Universal Robots PolyScope program: circle_run.urp

Program circle_run (installation=default directory=/programs/usbdisk createdIn=5.12.4.1101661 lastSavedIn=5.12.4.1101661)
Robot Program (runOnlyOnce=true)
  Script file /programs/usbdisk/circle.script
    | def draw_svg():
    |   draw_z = 0.074940
    |   # home
    |   movel(p[0.598550, -0.129200, 0.105150, 2.249000, -2.194000, 0.000000], a=0.8, v=0.25, r=0.0)
    |   # stroke 0 (form id 0): circle
    |   movel(p[0.452368, -0.119322, 0.118080, 2.230000, -2.212000, 0.000000], a=0.8, v=0.25, r=0.0)
    |   movep(p[0.452368, -0.119322, draw_z, 2.230000, -2.212000, 0.000000], a=0.5, v=0.02, r=0.001426)
    |   movep(p[0.452414, -0.116470, draw_z, 2.230000, -2.212000, 0.000000], a=0.5, v=0.02, r=0.002853)
    |   movep(p[0.452720, -0.110772, draw_z, 2.230000, -2.212000, 0.000000], a=0.5, v=0.02, r=0.002855)
    |   movep(p[0.453238, -0.105086, draw_z, 2.230000, -2.212000, 0.000000], a=0.5, v=0.02, r=0.002856)
    |   movep(p[0.453967, -0.099420, draw_z, 2.230000, -2.212000, 0.000000], a=0.5, v=0.02, r=0.002857)
    |   movep(p[0.454907, -0.093783, draw_z, 2.230000, -2.212000, 0.000000], a=0.5, v=0.02, r=0.002859)
    |   movep(p[0.456055, -0.088182, draw_z, 2.230000, -2.212000, 0.000000], a=0.5, v=0.02, r=0.002860)
    |   movep(p[0.457411, -0.082625, draw_z, 2.230000, -2.212000, 0.000000], a=0.5, v=0.02, r=0.002861)
    |   movep(p[0.458973, -0.077120, draw_z, 2.230000, -2.212000, 0.000000], a=0.5, v=0.02, r=0.002862)
    |   movep(p[0.460738, -0.071675, draw_z, 2.230000, -2.212000, 0.000000], a=0.5, v=0.02, r=0.002863)
    |   movep(p[0.462703, -0.066296, draw_z, 2.230000, -2.212000, 0.000000], a=0.5, v=0.02, r=0.002864)
    |   movep(p[0.464867, -0.060993, draw_z, 2.230000, -2.212000, 0.000000], a=0.5, v=0.02, r=0.002865)
    |   movep(p[0.467226, -0.055771, draw_z, 2.230000, -2.212000, 0.000000], a=0.5, v=0.02, r=0.002866)
    |   movep(p[0.469777, -0.050639, draw_z, 2.230000, -2.212000, 0.000000], a=0.5, v=0.02, r=0.002866)
    |   movep(p[0.472516, -0.045604, draw_z, 2.230000, -2.212000, 0.000000], a=0.5, v=0.02, r=0.002867)
    |   movep(p[0.475439, -0.040672, draw_z, 2.230000, -2.212000, 0.000000], a=0.5, v=0.02, r=0.002867)
    |   movep(p[0.478543, -0.035850, draw_z, 2.230000, -2.212000, 0.000000], a=0.5, v=0.02, r=0.002867)
    |   movep(p[0.481822, -0.031146, draw_z, 2.230000, -2.212000, 0.000000], a=0.5, v=0.02, r=0.002867)
    |   movep(p[0.485273, -0.026566, draw_z, 2.230000, -2.212000, 0.000000], a=0.5, v=0.02, r=0.002867)
    |   movep(p[0.488891, -0.022116, draw_z, 2.230000, -2.212000, 0.000000], a=0.5, v=0.02, r=0.002867)
    |   movep(p[0.492670, -0.017803, draw_z, 2.230000, -2.212000, 0.000000], a=0.5, v=0.02, r=0.002867)
    |   movep(p[0.496605, -0.013632, draw_z, 2.230000, -2.212000, 0.000000], a=0.5, v=0.02, r=0.002867)
    |   movep(p[0.500691, -0.009609, draw_z, 2.230000, -2.212000, 0.000000], a=0.5, v=0.02, r=0.002867)
    |   movep(p[0.504922, -0.005740, draw_z, 2.230000, -2.212000, 0.000000], a=0.5, v=0.02, r=0.002866)
    |   movep(p[0.509292, -0.002031, draw_z, 2.230000, -2.212000, 0.000000], a=0.5, v=0.02, r=0.002865)
    |   movep(p[0.513795, 0.001514, draw_z, 2.230000, -2.212000, 0.000000], a=0.5, v=0.02, r=0.002865)
    |   movep(p[0.518425, 0.004889, draw_z, 2.230000, -2.212000, 0.000000], a=0.5, v=0.02, r=0.002864)
    |   movep(p[0.523175, 0.008090, draw_z, 2.230000, -2.212000, 0.000000], a=0.5, v=0.02, r=0.002863)
    |   movep(p[0.528038, 0.011112, draw_z, 2.230000, -2.212000, 0.000000], a=0.5, v=0.02, r=0.002862)
    |   movep(p[0.533008, 0.013951, draw_z, 2.230000, -2.212000, 0.000000], a=0.5, v=0.02, r=0.002861)
    |   movep(p[0.538078, 0.016603, draw_z, 2.230000, -2.212000, 0.000000], a=0.5, v=0.02, r=0.002860)
    |   movep(p[0.543241, 0.019065, draw_z, 2.230000, -2.212000, 0.000000], a=0.5, v=0.02, r=0.002859)
    |   movep(p[0.548489, 0.021333, draw_z, 2.230000, -2.212000, 0.000000], a=0.5, v=0.02, r=0.002857)
    |   movep(p[0.553815, 0.023403, draw_z, 2.230000, -2.212000, 0.000000], a=0.5, v=0.02, r=0.002856)
    |   movep(p[0.559212, 0.025273, draw_z, 2.230000, -2.212000, 0.000000], a=0.5, v=0.02, r=0.002855)
    |   movep(p[0.564672, 0.026941, draw_z, 2.230000, -2.212000, 0.000000], a=0.5, v=0.02, r=0.002853)
    |   movep(p[0.570187, 0.028403, draw_z, 2.230000, -2.212000, 0.000000], a=0.5, v=0.02, r=0.002852)
    |   movep(p[0.575751, 0.029658, draw_z, 2.230000, -2.212000, 0.000000], a=0.5, v=0.02, r=0.002850)
    |   movep(p[0.581354, 0.030705, draw_z, 2.230000, -2.212000, 0.000000], a=0.5, v=0.02, r=0.002849)
    |   movep(p[0.586990, 0.031541, draw_z, 2.230000, -2.212000, 0.000000], a=0.5, v=0.02, r=0.002847)
    |   movep(p[0.592650, 0.032165, draw_z, 2.230000, -2.212000, 0.000000], a=0.5, v=0.02, r=0.002846)
    |   movep(p[0.598326, 0.032577, draw_z, 2.230000, -2.212000, 0.000000], a=0.5, v=0.02, r=0.002844)
    |   movep(p[0.604011, 0.032776, draw_z, 2.230000, -2.212000, 0.000000], a=0.5, v=0.02, r=0.002843)
    |   movep(p[0.609696, 0.032762, draw_z, 2.230000, -2.212000, 0.000000], a=0.5, v=0.02, r=0.002841)
    |   movep(p[0.615373, 0.032535, draw_z, 2.230000, -2.212000, 0.000000], a=0.5, v=0.02, r=0.002840)
    |   movep(p[0.621036, 0.032095, draw_z, 2.230000, -2.212000, 0.000000], a=0.5, v=0.02, r=0.002838)
    |   movep(p[0.626675, 0.031442, draw_z, 2.230000, -2.212000, 0.000000], a=0.5, v=0.02, r=0.002837)
    |   movep(p[0.632282, 0.030578, draw_z, 2.230000, -2.212000, 0.000000], a=0.5, v=0.02, r=0.002836)
    |   movep(p[0.637851, 0.029504, draw_z, 2.230000, -2.212000, 0.000000], a=0.5, v=0.02, r=0.002834)
    |   movep(p[0.643373, 0.028221, draw_z, 2.230000, -2.212000, 0.000000], a=0.5, v=0.02, r=0.002833)
    |   movep(p[0.648840, 0.026731, draw_z, 2.230000, -2.212000, 0.000000], a=0.5, v=0.02, r=0.002832)
    |   movep(p[0.654245, 0.025037, draw_z, 2.230000, -2.212000, 0.000000], a=0.5, v=0.02, r=0.002831)
    |   movep(p[0.659581, 0.023140, draw_z, 2.230000, -2.212000, 0.000000], a=0.5, v=0.02, r=0.002830)
    |   movep(p[0.664839, 0.021043, draw_z, 2.230000, -2.212000, 0.000000], a=0.5, v=0.02, r=0.002830)
    |   movep(p[0.670012, 0.018749, draw_z, 2.230000, -2.212000, 0.000000], a=0.5, v=0.02, r=0.002829)
    |   movep(p[0.675094, 0.016262, draw_z, 2.230000, -2.212000, 0.000000], a=0.5, v=0.02, r=0.002828)
    |   movep(p[0.680077, 0.013585, draw_z, 2.230000, -2.212000, 0.000000], a=0.5, v=0.02, r=0.002828)
    |   movep(p[0.684954, 0.010721, draw_z, 2.230000, -2.212000, 0.000000], a=0.5, v=0.02, r=0.002827)
    |   movep(p[0.689718, 0.007675, draw_z, 2.230000, -2.212000, 0.000000], a=0.5, v=0.02, r=0.002827)
    |   movep(p[0.694363, 0.004451, draw_z, 2.230000, -2.212000, 0.000000], a=0.5, v=0.02, r=0.002827)
    |   movep(p[0.698881, 0.001053, draw_z, 2.230000, -2.212000, 0.000000], a=0.5, v=0.02, r=0.002827)
    |   movep(p[0.703268, -0.002514, draw_z, 2.230000, -2.212000, 0.000000], a=0.5, v=0.02, r=0.002827)
    |   movep(p[0.707517, -0.006245, draw_z, 2.230000, -2.212000, 0.000000], a=0.5, v=0.02, r=0.002827)
    |   movep(p[0.711621, -0.010134, draw_z, 2.230000, -2.212000, 0.000000], a=0.5, v=0.02, r=0.002827)
    |   movep(p[0.715575, -0.014177, draw_z, 2.230000, -2.212000, 0.000000], a=0.5, v=0.02, r=0.002828)
    |   movep(p[0.719373, -0.018367, draw_z, 2.230000, -2.212000, 0.000000], a=0.5, v=0.02, r=0.002828)
    |   movep(p[0.723011, -0.022699, draw_z, 2.230000, -2.212000, 0.000000], a=0.5, v=0.02, r=0.002829)
    |   movep(p[0.726483, -0.027167, draw_z, 2.230000, -2.212000, 0.000000], a=0.5, v=0.02, r=0.002830)
    |   movep(p[0.729784, -0.031764, draw_z, 2.230000, -2.212000, 0.000000], a=0.5, v=0.02, r=0.002831)
    |   movep(p[0.732909, -0.036484, draw_z, 2.230000, -2.212000, 0.000000], a=0.5, v=0.02, r=0.002831)
    |   movep(p[0.735855, -0.041320, draw_z, 2.230000, -2.212000, 0.000000], a=0.5, v=0.02, r=0.002832)
    |   movep(p[0.738617, -0.046266, draw_z, 2.230000, -2.212000, 0.000000], a=0.5, v=0.02, r=0.002834)
    |   movep(p[0.741191, -0.051315, draw_z, 2.230000, -2.212000, 0.000000], a=0.5, v=0.02, r=0.002835)
    |   movep(p[0.743573, -0.056459, draw_z, 2.230000, -2.212000, 0.000000], a=0.5, v=0.02, r=0.002836)
    |   movep(p[0.745761, -0.061692, draw_z, 2.230000, -2.212000, 0.000000], a=0.5, v=0.02, r=0.002837)
    |   movep(p[0.747752, -0.067006, draw_z, 2.230000, -2.212000, 0.000000], a=0.5, v=0.02, r=0.002839)
    |   movep(p[0.749541, -0.072394, draw_z, 2.230000, -2.212000, 0.000000], a=0.5, v=0.02, r=0.002840)
    |   movep(p[0.751128, -0.077847, draw_z, 2.230000, -2.212000, 0.000000], a=0.5, v=0.02, r=0.002841)
    |   movep(p[0.752509, -0.083360, draw_z, 2.230000, -2.212000, 0.000000], a=0.5, v=0.02, r=0.002843)
    |   movep(p[0.753683, -0.088923, draw_z, 2.230000, -2.212000, 0.000000], a=0.5, v=0.02, r=0.002844)
    |   movep(p[0.754649, -0.094529, draw_z, 2.230000, -2.212000, 0.000000], a=0.5, v=0.02, r=0.002846)
    |   movep(p[0.755404, -0.100171, draw_z, 2.230000, -2.212000, 0.000000], a=0.5, v=0.02, r=0.002847)
    |   movep(p[0.755948, -0.105839, draw_z, 2.230000, -2.212000, 0.000000], a=0.5, v=0.02, r=0.002849)
    |   movep(p[0.756279, -0.111527, draw_z, 2.230000, -2.212000, 0.000000], a=0.5, v=0.02, r=0.002850)
    |   movep(p[0.756399, -0.117227, draw_z, 2.230000, -2.212000, 0.000000], a=0.5, v=0.02, r=0.002852)
    |   movep(p[0.756306, -0.122930, draw_z, 2.230000, -2.212000, 0.000000], a=0.5, v=0.02, r=0.002853)
    |   movep(p[0.756000, -0.128628, draw_z, 2.230000, -2.212000, 0.000000], a=0.5, v=0.02, r=0.002855)
    |   movep(p[0.755482, -0.134314, draw_z, 2.230000, -2.212000, 0.000000], a=0.5, v=0.02, r=0.002856)
    |   movep(p[0.754753, -0.139980, draw_z, 2.230000, -2.212000, 0.000000], a=0.5, v=0.02, r=0.002857)
    |   movep(p[0.753813, -0.145617, draw_z, 2.230000, -2.212000, 0.000000], a=0.5, v=0.02, r=0.002859)
    |   movep(p[0.752665, -0.151218, draw_z, 2.230000, -2.212000, 0.000000], a=0.5, v=0.02, r=0.002860)
    |   movep(p[0.751309, -0.156775, draw_z, 2.230000, -2.212000, 0.000000], a=0.5, v=0.02, r=0.002861)
    |   movep(p[0.749747, -0.162280, draw_z, 2.230000, -2.212000, 0.000000], a=0.5, v=0.02, r=0.002862)
    |   movep(p[0.747982, -0.167725, draw_z, 2.230000, -2.212000, 0.000000], a=0.5, v=0.02, r=0.002863)
    |   movep(p[0.746017, -0.173104, draw_z, 2.230000, -2.212000, 0.000000], a=0.5, v=0.02, r=0.002864)
    |   movep(p[0.743853, -0.178407, draw_z, 2.230000, -2.212000, 0.000000], a=0.5, v=0.02, r=0.002865)
    |   movep(p[0.741494, -0.183629, draw_z, 2.230000, -2.212000, 0.000000], a=0.5, v=0.02, r=0.002866)
    |   movep(p[0.738943, -0.188761, draw_z, 2.230000, -2.212000, 0.000000], a=0.5, v=0.02, r=0.002866)
    |   movep(p[0.736204, -0.193796, draw_z, 2.230000, -2.212000, 0.000000], a=0.5, v=0.02, r=0.002867)
    |   movep(p[0.733281, -0.198728, draw_z, 2.230000, -2.212000, 0.000000], a=0.5, v=0.02, r=0.002867)
    |   movep(p[0.730177, -0.203550, draw_z, 2.230000, -2.212000, 0.000000], a=0.5, v=0.02, r=0.002867)
    |   movep(p[0.726898, -0.208254, draw_z, 2.230000, -2.212000, 0.000000], a=0.5, v=0.02, r=0.002867)
    |   movep(p[0.723447, -0.212834, draw_z, 2.230000, -2.212000, 0.000000], a=0.5, v=0.02, r=0.002867)
    |   movep(p[0.719829, -0.217284, draw_z, 2.230000, -2.212000, 0.000000], a=0.5, v=0.02, r=0.002867)
    |   movep(p[0.716050, -0.221597, draw_z, 2.230000, -2.212000, 0.000000], a=0.5, v=0.02, r=0.002867)
    |   movep(p[0.712115, -0.225768, draw_z, 2.230000, -2.212000, 0.000000], a=0.5, v=0.02, r=0.002867)
    |   movep(p[0.708029, -0.229791, draw_z, 2.230000, -2.212000, 0.000000], a=0.5, v=0.02, r=0.002867)
    |   movep(p[0.703798, -0.233660, draw_z, 2.230000, -2.212000, 0.000000], a=0.5, v=0.02, r=0.002866)
    |   movep(p[0.699428, -0.237369, draw_z, 2.230000, -2.212000, 0.000000], a=0.5, v=0.02, r=0.002865)
    |   movep(p[0.694925, -0.240914, draw_z, 2.230000, -2.212000, 0.000000], a=0.5, v=0.02, r=0.002865)
    |   movep(p[0.690295, -0.244289, draw_z, 2.230000, -2.212000, 0.000000], a=0.5, v=0.02, r=0.002864)
    |   movep(p[0.685545, -0.247490, draw_z, 2.230000, -2.212000, 0.000000], a=0.5, v=0.02, r=0.002863)
    |   movep(p[0.680682, -0.250512, draw_z, 2.230000, -2.212000, 0.000000], a=0.5, v=0.02, r=0.002862)
    |   movep(p[0.675712, -0.253351, draw_z, 2.230000, -2.212000, 0.000000], a=0.5, v=0.02, r=0.002861)
    |   movep(p[0.670642, -0.256003, draw_z, 2.230000, -2.212000, 0.000000], a=0.5, v=0.02, r=0.002860)
    |   movep(p[0.665479, -0.258465, draw_z, 2.230000, -2.212000, 0.000000], a=0.5, v=0.02, r=0.002859)
    |   movep(p[0.660231, -0.260733, draw_z, 2.230000, -2.212000, 0.000000], a=0.5, v=0.02, r=0.002857)
    |   movep(p[0.654905, -0.262803, draw_z, 2.230000, -2.212000, 0.000000], a=0.5, v=0.02, r=0.002856)
    |   movep(p[0.649508, -0.264673, draw_z, 2.230000, -2.212000, 0.000000], a=0.5, v=0.02, r=0.002855)
    |   movep(p[0.644048, -0.266341, draw_z, 2.230000, -2.212000, 0.000000], a=0.5, v=0.02, r=0.002853)
    |   movep(p[0.638533, -0.267803, draw_z, 2.230000, -2.212000, 0.000000], a=0.5, v=0.02, r=0.002852)
    |   movep(p[0.632969, -0.269058, draw_z, 2.230000, -2.212000, 0.000000], a=0.5, v=0.02, r=0.002850)
    |   movep(p[0.627366, -0.270105, draw_z, 2.230000, -2.212000, 0.000000], a=0.5, v=0.02, r=0.002849)
    |   movep(p[0.621730, -0.270941, draw_z, 2.230000, -2.212000, 0.000000], a=0.5, v=0.02, r=0.002847)
    |   movep(p[0.616070, -0.271565, draw_z, 2.230000, -2.212000, 0.000000], a=0.5, v=0.02, r=0.002846)
    |   movep(p[0.610394, -0.271977, draw_z, 2.230000, -2.212000, 0.000000], a=0.5, v=0.02, r=0.002844)
    |   movep(p[0.604709, -0.272176, draw_z, 2.230000, -2.212000, 0.000000], a=0.5, v=0.02, r=0.002843)
    |   movep(p[0.599024, -0.272162, draw_z, 2.230000, -2.212000, 0.000000], a=0.5, v=0.02, r=0.002841)
    |   movep(p[0.593347, -0.271935, draw_z, 2.230000, -2.212000, 0.000000], a=0.5, v=0.02, r=0.002840)
    |   movep(p[0.587684, -0.271495, draw_z, 2.230000, -2.212000, 0.000000], a=0.5, v=0.02, r=0.002838)
    |   movep(p[0.582045, -0.270842, draw_z, 2.230000, -2.212000, 0.000000], a=0.5, v=0.02, r=0.002837)
    |   movep(p[0.576438, -0.269978, draw_z, 2.230000, -2.212000, 0.000000], a=0.5, v=0.02, r=0.002836)
    |   movep(p[0.570869, -0.268904, draw_z, 2.230000, -2.212000, 0.000000], a=0.5, v=0.02, r=0.002834)
    |   movep(p[0.565347, -0.267621, draw_z, 2.230000, -2.212000, 0.000000], a=0.5, v=0.02, r=0.002833)
    |   movep(p[0.559880, -0.266131, draw_z, 2.230000, -2.212000, 0.000000], a=0.5, v=0.02, r=0.002832)
    |   movep(p[0.554475, -0.264437, draw_z, 2.230000, -2.212000, 0.000000], a=0.5, v=0.02, r=0.002831)
    |   movep(p[0.549139, -0.262540, draw_z, 2.230000, -2.212000, 0.000000], a=0.5, v=0.02, r=0.002830)
    |   movep(p[0.543881, -0.260443, draw_z, 2.230000, -2.212000, 0.000000], a=0.5, v=0.02, r=0.002830)
    |   movep(p[0.538708, -0.258149, draw_z, 2.230000, -2.212000, 0.000000], a=0.5, v=0.02, r=0.002829)
    |   movep(p[0.533626, -0.255662, draw_z, 2.230000, -2.212000, 0.000000], a=0.5, v=0.02, r=0.002828)
    |   movep(p[0.528643, -0.252985, draw_z, 2.230000, -2.212000, 0.000000], a=0.5, v=0.02, r=0.002828)
    |   movep(p[0.523766, -0.250121, draw_z, 2.230000, -2.212000, 0.000000], a=0.5, v=0.02, r=0.002827)
    |   movep(p[0.519002, -0.247075, draw_z, 2.230000, -2.212000, 0.000000], a=0.5, v=0.02, r=0.002827)
    |   movep(p[0.514357, -0.243851, draw_z, 2.230000, -2.212000, 0.000000], a=0.5, v=0.02, r=0.002827)
    |   movep(p[0.509839, -0.240453, draw_z, 2.230000, -2.212000, 0.000000], a=0.5, v=0.02, r=0.002827)
    |   movep(p[0.505452, -0.236886, draw_z, 2.230000, -2.212000, 0.000000], a=0.5, v=0.02, r=0.002827)
    |   movep(p[0.501203, -0.233155, draw_z, 2.230000, -2.212000, 0.000000], a=0.5, v=0.02, r=0.002827)
    |   movep(p[0.497099, -0.229266, draw_z, 2.230000, -2.212000, 0.000000], a=0.5, v=0.02, r=0.002827)
    |   movep(p[0.493145, -0.225223, draw_z, 2.230000, -2.212000, 0.000000], a=0.5, v=0.02, r=0.002828)
    |   movep(p[0.489347, -0.221033, draw_z, 2.230000, -2.212000, 0.000000], a=0.5, v=0.02, r=0.002828)
    |   movep(p[0.485709, -0.216701, draw_z, 2.230000, -2.212000, 0.000000], a=0.5, v=0.02, r=0.002829)
    |   movep(p[0.482237, -0.212233, draw_z, 2.230000, -2.212000, 0.000000], a=0.5, v=0.02, r=0.002830)
    |   movep(p[0.478936, -0.207636, draw_z, 2.230000, -2.212000, 0.000000], a=0.5, v=0.02, r=0.002831)
    |   movep(p[0.475811, -0.202916, draw_z, 2.230000, -2.212000, 0.000000], a=0.5, v=0.02, r=0.002831)
    |   movep(p[0.472865, -0.198080, draw_z, 2.230000, -2.212000, 0.000000], a=0.5, v=0.02, r=0.002832)
    |   movep(p[0.470103, -0.193134, draw_z, 2.230000, -2.212000, 0.000000], a=0.5, v=0.02, r=0.002834)
    |   movep(p[0.467529, -0.188085, draw_z, 2.230000, -2.212000, 0.000000], a=0.5, v=0.02, r=0.002835)
    |   movep(p[0.465147, -0.182941, draw_z, 2.230000, -2.212000, 0.000000], a=0.5, v=0.02, r=0.002836)
    |   movep(p[0.462959, -0.177708, draw_z, 2.230000, -2.212000, 0.000000], a=0.5, v=0.02, r=0.002837)
    |   movep(p[0.460968, -0.172394, draw_z, 2.230000, -2.212000, 0.000000], a=0.5, v=0.02, r=0.002839)
    |   movep(p[0.459179, -0.167006, draw_z, 2.230000, -2.212000, 0.000000], a=0.5, v=0.02, r=0.002840)
    |   movep(p[0.457592, -0.161553, draw_z, 2.230000, -2.212000, 0.000000], a=0.5, v=0.02, r=0.002841)
    |   movep(p[0.456211, -0.156040, draw_z, 2.230000, -2.212000, 0.000000], a=0.5, v=0.02, r=0.002843)
    |   movep(p[0.455037, -0.150477, draw_z, 2.230000, -2.212000, 0.000000], a=0.5, v=0.02, r=0.002844)
    |   movep(p[0.454071, -0.144871, draw_z, 2.230000, -2.212000, 0.000000], a=0.5, v=0.02, r=0.002846)
    |   movep(p[0.453316, -0.139229, draw_z, 2.230000, -2.212000, 0.000000], a=0.5, v=0.02, r=0.002847)
    |   movep(p[0.452772, -0.133561, draw_z, 2.230000, -2.212000, 0.000000], a=0.5, v=0.02, r=0.002849)
    |   movep(p[0.452441, -0.127873, draw_z, 2.230000, -2.212000, 0.000000], a=0.5, v=0.02, r=0.002850)
    |   movep(p[0.452321, -0.122173, draw_z, 2.230000, -2.212000, 0.000000], a=0.5, v=0.02, r=0.001426)
    |   movep(p[0.452368, -0.119322, draw_z, 2.230000, -2.212000, 0.000000], a=0.5, v=0.02, r=0.000000)
    |   movel(p[0.452368, -0.119322, 0.118080, 2.230000, -2.212000, 0.000000], a=0.8, v=0.25, r=0.0)
    |   # park
    |   movel(p[0.598550, -0.129200, 0.105150, 2.249000, -2.194000, 0.000000], a=0.8, v=0.25, r=0.0)
    | end
    | draw_svg()
